(* IEC 61131-3 sources: programs/VI-54/VI-54_20171205/VI-54_20171205/Stations/PLC_VI54/VI-54_171014/Class/FilterIFCsignal, 1 file *)

(* ---- FilterIFCsignal.st ---- *)
(*!
<Class
	Name               = "FilterIFCsignal"
	Revision           = "1.0"
	RealtimeTask       = "false"
	CyclicTask         = "false"
	BackgroundTask     = "false"
	Sigmatek           = "false"
	OSInterface        = "false"
	HighPriority       = "false"
	Automatic          = "false"
	UpdateMode         = "Prescan"
	SharedCommandTable = "true"
	Objectsize         = "(570,240)">
	<Channels>
		<Server Name="TriggerFilter" Visualized="true" Initialize="false" WriteProtected="true" Retentive="false"/>
		<Client Name="iFilterTime" Required="false" Internal="false"/>
		<Client Name="iMaskTime" Required="false" Internal="false"/>
		<Client Name="iTrigger" Required="false" Internal="false"/>
		<Client Name="Saved_FilterTime" Required="true" Internal="true"/>
		<Client Name="Saved_LineSpeed" Required="true" Internal="true"/>
		<Client Name="Saved_MaskTime" Required="true" Internal="true"/>
		<Client Name="STD" Required="true" Internal="true"/>
	</Channels>
	<Network Name="FilterIFCsignal">
		<!-- List of Components in this network -->
		<Components>
			<Object
				Name       = "Saved_FilterTime"
				Class      = "Ram"
				Position   = "(270,540)"
				Visualized = "true"
				Remotely   = "true">
				<Channels>
					<Server Name="Data"/>
				</Channels>
			</Object>
			<Object
				Name       = "Saved_LineSpeed"
				Class      = "Ram"
				Position   = "(270,390)"
				Visualized = "true"
				Remotely   = "true">
				<Channels>
					<Server Name="Data"/>
				</Channels>
			</Object>
			<Object
				Name       = "Saved_MaskTime"
				Class      = "Ram"
				Position   = "(270,690)"
				Visualized = "true"
				Remotely   = "true">
				<Channels>
					<Server Name="Data"/>
				</Channels>
			</Object>
			<Object
				Name           = "STD"
				Class          = "Standard"
				Position       = "(270,240)"
				Visualized     = "false"
				BackgroundTime = "1000 ms">
				<Channels>
					<Server Name="ClassSvr"/>
				</Channels>
			</Object>
		</Components>
		<Comments>
		</Comments>
		<!-- List of Connections in this network -->
		<Connections>
			<Connection Source="this.STD" Destination="STD.ClassSvr"/>
			<Connection Source="this.Saved_LineSpeed" Destination="Saved_LineSpeed.Data"/>
			<Connection Source="this.Saved_FilterTime" Destination="Saved_FilterTime.Data"/>
			<Connection Source="this.Saved_MaskTime" Destination="Saved_MaskTime.Data"/>
		</Connections>
		<!-- Headerfiles -->
		<Options>
		</Options>
	</Network>
</Class>
*)
FilterIFCsignal : CLASS
  //Servers:
	TriggerFilter 	: SvrChCmd_DINT;
  //Clients:
	iTrigger 	: CltCh_DINT;
	STD 	: CltChCmd_Standard;
	iMaskTime 	: CltCh_DINT;
	iFilterTime 	: CltCh_DINT;
	Saved_LineSpeed 	: CltChCmd_Ram;
	Saved_FilterTime 	: CltChCmd_Ram;
	Saved_MaskTime 	: CltChCmd_Ram;
  //Variables:
		udFilterTime 	: UDINT;
		MaskTime 	: DINT;
		LineSpeed 	: REAL;
		DistanceFilterTime 	: REAL;
		NewFilterTime 	: DINT;
		DistanceMaskTime 	: REAL;
		NewMaskTime 	: DINT;
  //Functions:

	FUNCTION GLOBAL SetLineSpeed
		VAR_INPUT
			Speed 	: DINT;
		END_VAR;

	FUNCTION VIRTUAL GLOBAL TriggerFilter::Read
		VAR_OUTPUT
			output (EAX) 	: DINT;
		END_VAR;
  //Tables:
	FUNCTION @STD
		VAR_OUTPUT
			ret_code	: CONFSTATES;
		END_VAR;
	FUNCTION GLOBAL TAB @CT_;
END_CLASS;

#pragma using Ram
#pragma using Standard

FUNCTION VIRTUAL GLOBAL FilterIFCsignal::TriggerFilter::Read
	VAR_OUTPUT
		output (EAX) 	: DINT;
	END_VAR

  // Read inputs
  iTrigger    := iTrigger.Read();
  iMaskTime   := iMaskTime.Read();
  iFilterTime := iFilterTime.Read();

  // Save changes
  if iFilterTime <> Saved_FilterTime.Read() then
    Saved_FilterTime.Write(input:= iFilterTime);
    Saved_LineSpeed.Write(input:= to_dint LineSpeed);
  elsif iMaskTime <> Saved_MaskTime.Read() then
    Saved_MaskTime.Write(input:= iMaskTime);
    Saved_LineSpeed.Write(input:= to_dint LineSpeed);
  elsif (LineSpeed <> Saved_LineSpeed.Read()) & (LineSpeed > 10) then // Change filter and mask time, only when speed is higher than 1.0 m/min
    DistanceFilterTime := (to_real iFilterTime * Saved_LineSpeed.Read());
    NewFilterTime      := to_dint(DistanceFilterTime / to_real LineSpeed);

    DistanceMaskTime   := (to_real iMaskTime * Saved_LineSpeed.Read());
    NewMaskTime        := to_dint(DistanceMaskTime / to_real LineSpeed);

    Saved_FilterTime.Write(input:= NewFilterTime);
    iFilterTime.Write(input:= NewFilterTime);
    Saved_MaskTime.Write(input:= NewMaskTime);
    iMaskTime.Write(input:= NewMaskTime);
    Saved_LineSpeed.Write(input:= to_dint LineSpeed);
  end_if;

  // filtertijd
  // Het product moet een minimale tijdsduur hoog zijn voordat het pas echt een puls wordt
  // Anders is het vuil / afval
  if iTrigger = 1 then
    if (ops.tAbsolute - udFilterTime) >= to_udint(iFilterTime) then
      TriggerFilter := 1;
    end_if;
  else
    udFilterTime := ops.tAbsolute;
  end_if;

  // minimaal hooghouden van signaal
  if iMaskTime <= 100 then
    MaskTime := 100;
  else
    MaskTime := iMaskTime;
  end_if;
  if STD.TON(IN:= TriggerFilter, PT:= MaskTime) then // hou 100ms hoog
    TriggerFilter := 0;
  end_if;

	output := TriggerFilter;

END_FUNCTION

FUNCTION GLOBAL FilterIFCsignal::SetLineSpeed
	VAR_INPUT
		Speed 	: DINT;
	END_VAR

  LineSpeed := (to_real Speed ToMperMin);

END_FUNCTION
